// TIA Portal V20 export
FUNCTION_BLOCK "LER_InspectionInterface"   // FB50060, LAD
// stored: Access Published, MemoryReserve 100, SetENOAutomatically false
   VAR_INPUT
      Clamped : Bool;
      UnClamped : Bool;
      Celldetect : Bool;
      DryRun : Bool;
      SoftCam_X : "LER_typeSoftCamInterface";   // [6] Avoid , [7] Inst contac,[1]Ready
      SoftCam_Z : "LER_typeSoftCamInterface";   // [1] Ready , Avoid
      SoftCAm_C : "LER_typeSoftCamInterface";
      ProductionTimeTriger : Bool;
      Part_ID : String[32];
   END_VAR
   VAR_OUTPUT
      Axis_DisChargePositionLock : Bool;
      Axis_DisChargePositionCmd : Bool;   // for AutoSeq
      Axis_AvoidPositionCmd : Bool;   // for AutoSeq
      Axis_LoadComeplte : Bool;
      Insp_Req_Unclamp : Bool;   // for AutoSeq
   END_VAR
   VAR_IN_OUT
      BA60 : "LER_typeCommunicationInspection";
   END_VAR
   VAR
      DTL : DTL;
      STKtoINSP_Log : Array[0..50] of "LER_typeCommonDataInspection";
      P : Array[0..15] of Bool;
      Logic : Struct
         "a" : Bool;
         "b" : Bool;
      END_STRUCT;
      CleanData : "LER_typeCommonDataInspection";
   END_VAR
   VAR_TEMP
      REt : Int;
   END_VAR
   VAR_TEMP   // added for the SCL form of the ladder/FBD networks
      _w1 : Bool;
   END_VAR
BEGIN

REGION Network 2
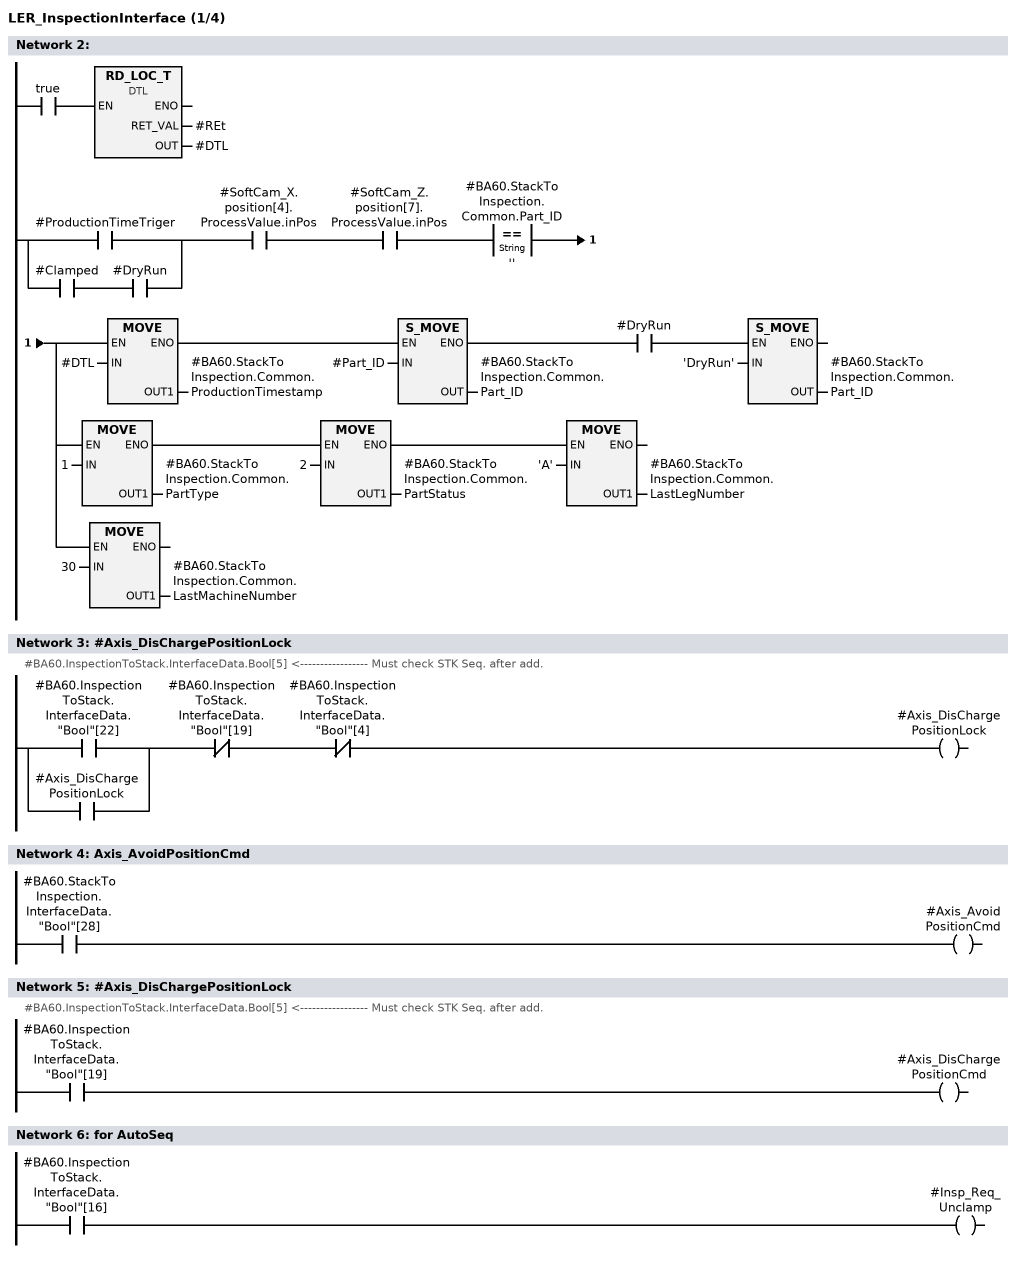
   RUNG wire#powerrail
      Contact( true )
      { S7_Templates := "date_type := DTL" } RD_LOC_T(RET_VAL => #REt, OUT => #DTL)
   END_RUNG
   RUNG wire#powerrail
      Contact( #ProductionTimeTriger )
      wire#w1
      Contact( #SoftCam_X.position[4].ProcessValue.inPos )
      Contact( #SoftCam_Z.position[7].ProcessValue.inPos )
      { S7_Templates := "SrcType := String" } EQ_Contact(in1 := #BA60.StackToInspection.Common.Part_ID, in2 := '')
      wire#w2
      Move(in := #DTL, out1 => #BA60.StackToInspection.Common.ProductionTimestamp)
      S_Move(in := #Part_ID, out => #BA60.StackToInspection.Common.Part_ID)
      Contact( #DryRun )
      S_Move(in := 'DryRun', out => #BA60.StackToInspection.Common.Part_ID)
   END_RUNG
   RUNG wire#powerrail
      Contact( #Clamped )
      Contact( #DryRun )
   END_RUNG wire#w1
   RUNG wire#w2
      Move(in := 1, out1 => #BA60.StackToInspection.Common.PartType)
      Move(in := 2, out1 => #BA60.StackToInspection.Common.PartStatus)
      Move(in := 'A', out1 => #BA60.StackToInspection.Common.LastLegNumber)
   END_RUNG
   RUNG wire#w2
      Move(in := 30, out1 => #BA60.StackToInspection.Common.LastMachineNumber)
   END_RUNG
   // the same network as SCL:
   IF true THEN #REt := RD_LOC_T(OUT => #DTL); END_IF;
   #_w1 := (#ProductionTimeTriger OR (#Clamped AND #DryRun)) AND #SoftCam_X.position[4].ProcessValue.inPos AND #SoftCam_Z.position[7].ProcessValue.inPos AND (#BA60.StackToInspection.Common.Part_ID = '');
   IF #_w1 THEN
       #BA60.StackToInspection.Common.ProductionTimestamp := #DTL;
       #BA60.StackToInspection.Common.Part_ID := #Part_ID;
   END_IF;
   IF #_w1 AND #DryRun THEN #BA60.StackToInspection.Common.Part_ID := 'DryRun'; END_IF;
   IF #_w1 THEN
       #BA60.StackToInspection.Common.PartType := 1;
       #BA60.StackToInspection.Common.PartStatus := 2;
       #BA60.StackToInspection.Common.LastLegNumber := 'A';
       #BA60.StackToInspection.Common.LastMachineNumber := 30;
   END_IF;
END_REGION

REGION Network 3: #Axis_DisChargePositionLock
   // #BA60.InspectionToStack.InterfaceData.Bool[5] <----------------- Must check STK Seq. after add.
   RUNG wire#powerrail
      Contact( #BA60.InspectionToStack.InterfaceData."Bool"[22] )
      wire#w1
      I_Contact( #BA60.InspectionToStack.InterfaceData."Bool"[19] )
      I_Contact( #BA60.InspectionToStack.InterfaceData."Bool"[4] )
      Coil( #Axis_DisChargePositionLock )
   END_RUNG
   RUNG wire#powerrail
      Contact( #Axis_DisChargePositionLock )
   END_RUNG wire#w1
   // the same network as SCL:
   #Axis_DisChargePositionLock := (#BA60.InspectionToStack.InterfaceData."Bool"[22] OR #Axis_DisChargePositionLock) AND NOT #BA60.InspectionToStack.InterfaceData."Bool"[19] AND NOT #BA60.InspectionToStack.InterfaceData."Bool"[4];
END_REGION

REGION Network 4: Axis_AvoidPositionCmd
   RUNG wire#powerrail
      Contact( #BA60.StackToInspection.InterfaceData."Bool"[28] )
      Coil( #Axis_AvoidPositionCmd )
   END_RUNG
   // the same network as SCL:
   #Axis_AvoidPositionCmd := #BA60.StackToInspection.InterfaceData."Bool"[28];
END_REGION

REGION Network 5: #Axis_DisChargePositionLock
   // #BA60.InspectionToStack.InterfaceData.Bool[5] <----------------- Must check STK Seq. after add.
   RUNG wire#powerrail
      Contact( #BA60.InspectionToStack.InterfaceData."Bool"[19] )
      Coil( #Axis_DisChargePositionCmd )
   END_RUNG
   // the same network as SCL:
   #Axis_DisChargePositionCmd := #BA60.InspectionToStack.InterfaceData."Bool"[19];
END_REGION

REGION Network 6: for AutoSeq
   RUNG wire#powerrail
      Contact( #BA60.InspectionToStack.InterfaceData."Bool"[16] )
      Coil( #Insp_Req_Unclamp )
   END_RUNG
   // the same network as SCL:
   #Insp_Req_Unclamp := #BA60.InspectionToStack.InterfaceData."Bool"[16];
END_REGION

REGION Network 7: for AutoSeq - Load Complete
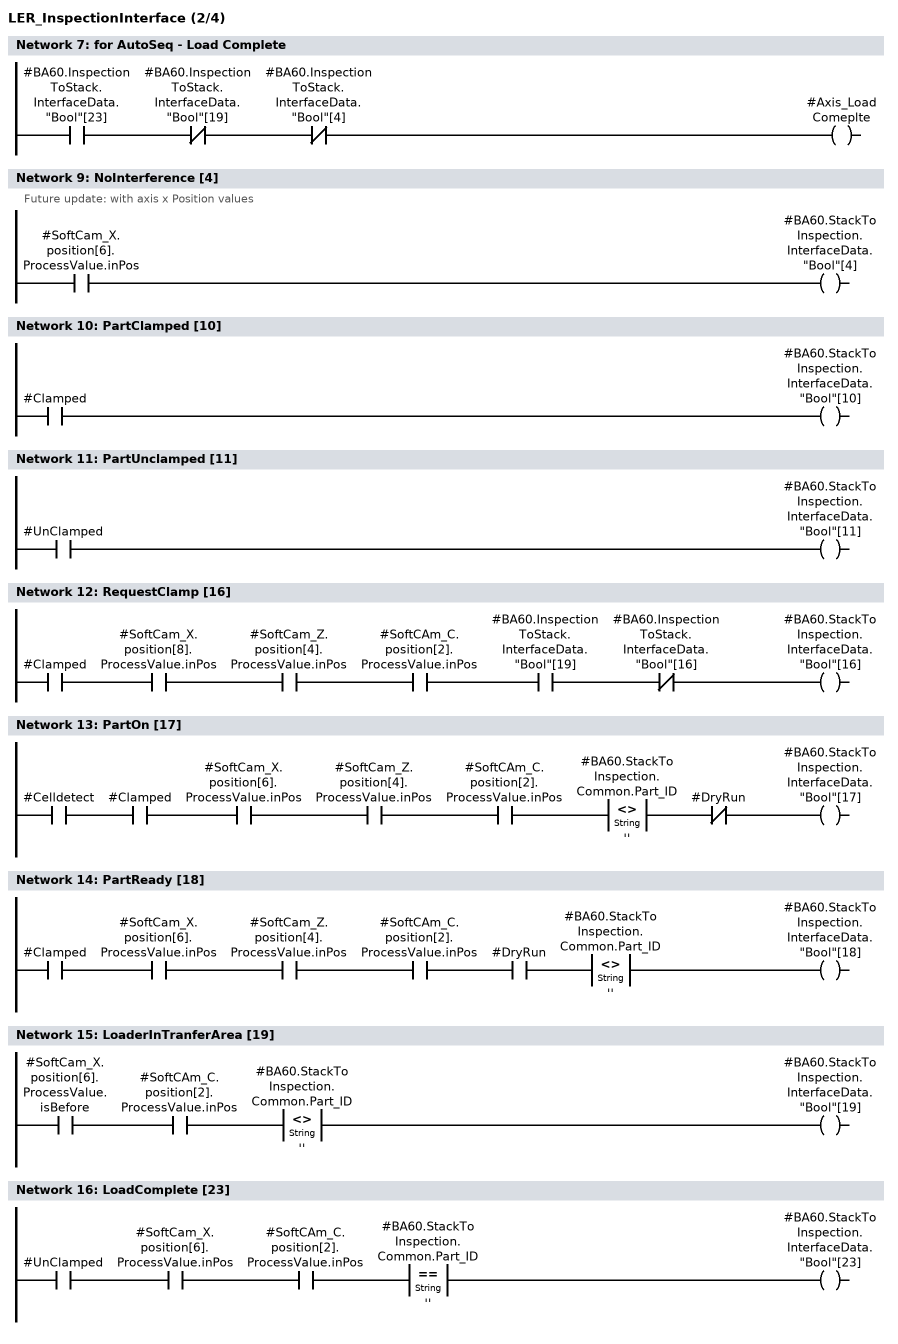
   RUNG wire#powerrail
      Contact( #BA60.InspectionToStack.InterfaceData."Bool"[23] )
      I_Contact( #BA60.InspectionToStack.InterfaceData."Bool"[19] )
      I_Contact( #BA60.InspectionToStack.InterfaceData."Bool"[4] )
      Coil( #Axis_LoadComeplte )
   END_RUNG
   // the same network as SCL:
   #Axis_LoadComeplte := #BA60.InspectionToStack.InterfaceData."Bool"[23] AND NOT #BA60.InspectionToStack.InterfaceData."Bool"[19] AND NOT #BA60.InspectionToStack.InterfaceData."Bool"[4];
END_REGION

REGION Network 8: ========================= Inspection To Stack ===================================
END_REGION

REGION Network 9: NoInterference [4]
   // Future update: with axis x Position values
   RUNG wire#powerrail
      Contact( #SoftCam_X.position[6].ProcessValue.inPos )
      Coil( #BA60.StackToInspection.InterfaceData."Bool"[4] )
   END_RUNG
   // the same network as SCL:
   #BA60.StackToInspection.InterfaceData."Bool"[4] := #SoftCam_X.position[6].ProcessValue.inPos;
END_REGION

REGION Network 10: PartClamped [10]
   RUNG wire#powerrail
      Contact( #Clamped )
      Coil( #BA60.StackToInspection.InterfaceData."Bool"[10] )
   END_RUNG
   // the same network as SCL:
   #BA60.StackToInspection.InterfaceData."Bool"[10] := #Clamped;
END_REGION

REGION Network 11: PartUnclamped [11]
   RUNG wire#powerrail
      Contact( #UnClamped )
      Coil( #BA60.StackToInspection.InterfaceData."Bool"[11] )
   END_RUNG
   // the same network as SCL:
   #BA60.StackToInspection.InterfaceData."Bool"[11] := #UnClamped;
END_REGION

REGION Network 12: RequestClamp [16]
   RUNG wire#powerrail
      Contact( #Clamped )
      Contact( #SoftCam_X.position[8].ProcessValue.inPos )
      Contact( #SoftCam_Z.position[4].ProcessValue.inPos )
      Contact( #SoftCAm_C.position[2].ProcessValue.inPos )
      Contact( #BA60.InspectionToStack.InterfaceData."Bool"[19] )
      I_Contact( #BA60.InspectionToStack.InterfaceData."Bool"[16] )
      Coil( #BA60.StackToInspection.InterfaceData."Bool"[16] )
   END_RUNG
   // the same network as SCL:
   #BA60.StackToInspection.InterfaceData."Bool"[16] := #Clamped AND #SoftCam_X.position[8].ProcessValue.inPos AND #SoftCam_Z.position[4].ProcessValue.inPos AND #SoftCAm_C.position[2].ProcessValue.inPos AND #BA60.InspectionToStack.InterfaceData."Bool"[19] AND NOT #BA60.InspectionToStack.InterfaceData."Bool"[16];
END_REGION

REGION Network 13: PartOn [17]
   RUNG wire#powerrail
      Contact( #Celldetect )
      Contact( #Clamped )
      Contact( #SoftCam_X.position[6].ProcessValue.inPos )
      Contact( #SoftCam_Z.position[4].ProcessValue.inPos )
      Contact( #SoftCAm_C.position[2].ProcessValue.inPos )
      { S7_Templates := "SrcType := String" } NE_Contact(in1 := #BA60.StackToInspection.Common.Part_ID, in2 := '')
      I_Contact( #DryRun )
      Coil( #BA60.StackToInspection.InterfaceData."Bool"[17] )
   END_RUNG
   // the same network as SCL:
   #BA60.StackToInspection.InterfaceData."Bool"[17] := #Celldetect AND #Clamped AND #SoftCam_X.position[6].ProcessValue.inPos AND #SoftCam_Z.position[4].ProcessValue.inPos AND #SoftCAm_C.position[2].ProcessValue.inPos AND (#BA60.StackToInspection.Common.Part_ID <> '') AND NOT #DryRun;
END_REGION

REGION Network 14: PartReady [18]
   RUNG wire#powerrail
      Contact( #Clamped )
      Contact( #SoftCam_X.position[6].ProcessValue.inPos )
      Contact( #SoftCam_Z.position[4].ProcessValue.inPos )
      Contact( #SoftCAm_C.position[2].ProcessValue.inPos )
      Contact( #DryRun )
      { S7_Templates := "SrcType := String" } NE_Contact(in1 := #BA60.StackToInspection.Common.Part_ID, in2 := '')
      Coil( #BA60.StackToInspection.InterfaceData."Bool"[18] )
   END_RUNG
   // the same network as SCL:
   #BA60.StackToInspection.InterfaceData."Bool"[18] := #Clamped AND #SoftCam_X.position[6].ProcessValue.inPos AND #SoftCam_Z.position[4].ProcessValue.inPos AND #SoftCAm_C.position[2].ProcessValue.inPos AND #DryRun AND (#BA60.StackToInspection.Common.Part_ID <> '');
END_REGION

REGION Network 15: LoaderInTranferArea [19]
   RUNG wire#powerrail
      Contact( #SoftCam_X.position[6].ProcessValue.isBefore )
      Contact( #SoftCAm_C.position[2].ProcessValue.inPos )
      { S7_Templates := "SrcType := String" } NE_Contact(in1 := #BA60.StackToInspection.Common.Part_ID, in2 := '')
      Coil( #BA60.StackToInspection.InterfaceData."Bool"[19] )
   END_RUNG
   // the same network as SCL:
   #BA60.StackToInspection.InterfaceData."Bool"[19] := #SoftCam_X.position[6].ProcessValue.isBefore AND #SoftCAm_C.position[2].ProcessValue.inPos AND (#BA60.StackToInspection.Common.Part_ID <> '');
END_REGION

REGION Network 16: LoadComplete [23]
   RUNG wire#powerrail
      Contact( #UnClamped )
      Contact( #SoftCam_X.position[6].ProcessValue.inPos )
      Contact( #SoftCAm_C.position[2].ProcessValue.inPos )
      { S7_Templates := "SrcType := String" } EQ_Contact(in1 := #BA60.StackToInspection.Common.Part_ID, in2 := '')
      Coil( #BA60.StackToInspection.InterfaceData."Bool"[23] )
   END_RUNG
   // the same network as SCL:
   #BA60.StackToInspection.InterfaceData."Bool"[23] := #UnClamped AND #SoftCam_X.position[6].ProcessValue.inPos AND #SoftCAm_C.position[2].ProcessValue.inPos AND (#BA60.StackToInspection.Common.Part_ID = '');
END_REGION

REGION Network 17: DataCatchUp [26]
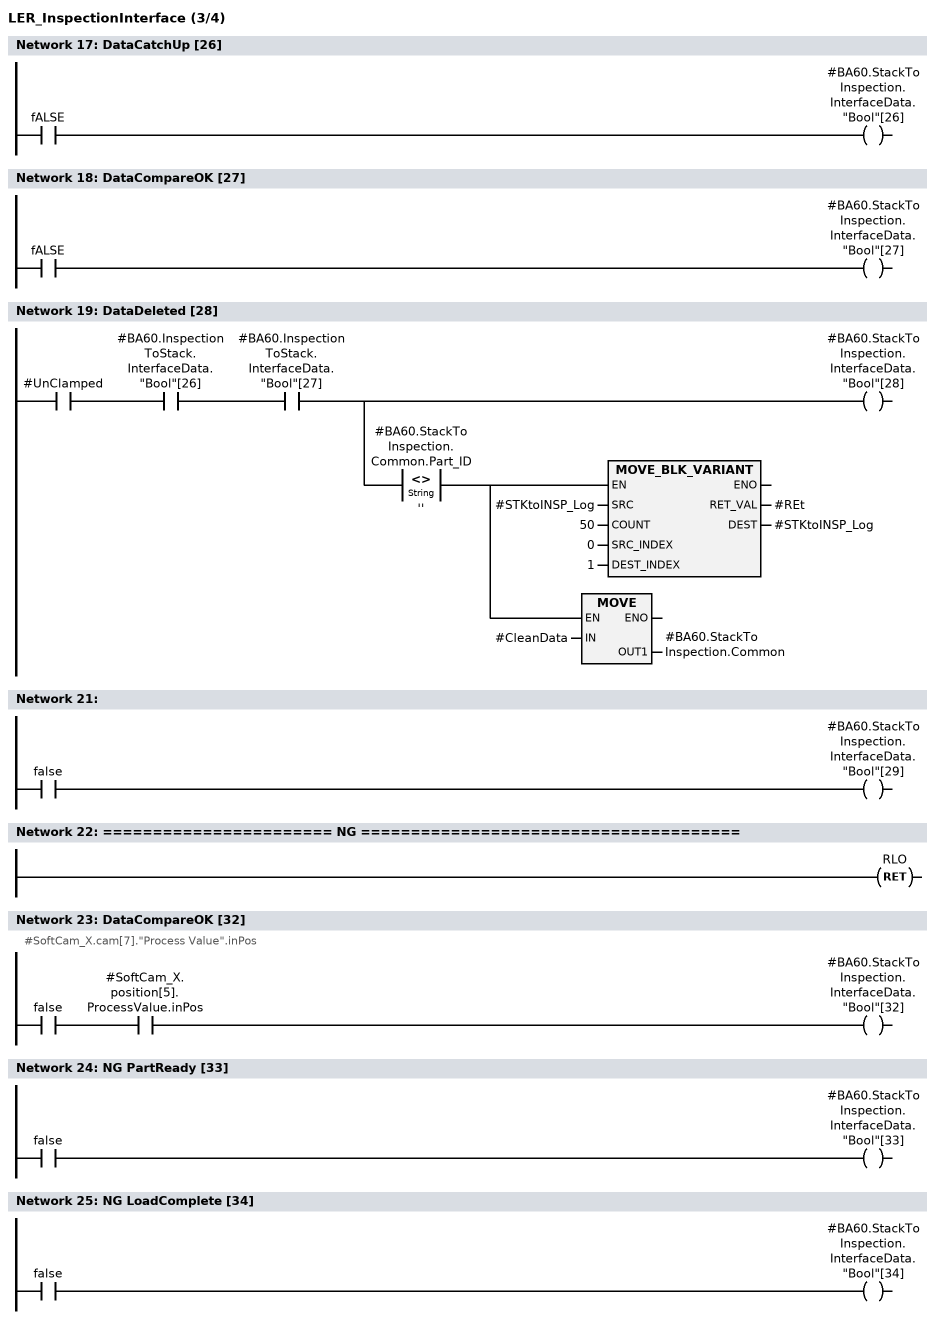
   RUNG wire#powerrail
      Contact( fALSE )
      Coil( #BA60.StackToInspection.InterfaceData."Bool"[26] )
   END_RUNG
   // the same network as SCL:
   #BA60.StackToInspection.InterfaceData."Bool"[26] := fALSE;
END_REGION

REGION Network 18: DataCompareOK [27]
   RUNG wire#powerrail
      Contact( fALSE )
      Coil( #BA60.StackToInspection.InterfaceData."Bool"[27] )
   END_RUNG
   // the same network as SCL:
   #BA60.StackToInspection.InterfaceData."Bool"[27] := fALSE;
END_REGION

REGION Network 19: DataDeleted [28]
   RUNG wire#powerrail
      Contact( #UnClamped )
      Contact( #BA60.InspectionToStack.InterfaceData."Bool"[26] )
      Contact( #BA60.InspectionToStack.InterfaceData."Bool"[27] )
      wire#w1
      Coil( #BA60.StackToInspection.InterfaceData."Bool"[28] )
   END_RUNG
   RUNG wire#w1
      { S7_Templates := "SrcType := String" } NE_Contact(in1 := #BA60.StackToInspection.Common.Part_ID, in2 := '')
      wire#w2
      MOVE_BLK_VARIANT(SRC := #STKtoINSP_Log, COUNT := 50, SRC_INDEX := 0, DEST_INDEX := 1, Ret_Val => #REt, DEST => #STKtoINSP_Log)
   END_RUNG
   RUNG wire#w2
      Move(in := #CleanData, out1 => #BA60.StackToInspection.Common)
   END_RUNG
   // the same network as SCL:
   #BA60.StackToInspection.InterfaceData."Bool"[28] := #UnClamped AND #BA60.InspectionToStack.InterfaceData."Bool"[26] AND #BA60.InspectionToStack.InterfaceData."Bool"[27];
   IF #UnClamped AND #BA60.InspectionToStack.InterfaceData."Bool"[26] AND #BA60.InspectionToStack.InterfaceData."Bool"[27] AND (#BA60.StackToInspection.Common.Part_ID <> '') THEN
       #REt := MOVE_BLK_VARIANT(SRC := #STKtoINSP_Log,
                               COUNT := 50,
                               SRC_INDEX := 0,
                               DEST_INDEX := 1,
                               DEST => #STKtoINSP_Log);
       #BA60.StackToInspection.Common := #CleanData;
   END_IF;
END_REGION

REGION Network 21
   RUNG wire#powerrail
      Contact( false )
      Coil( #BA60.StackToInspection.InterfaceData."Bool"[29] )
   END_RUNG
   // the same network as SCL:
   #BA60.StackToInspection.InterfaceData."Bool"[29] := false;
END_REGION

REGION Network 22: ======================= NG ======================================
   ENO := TRUE;
   RETURN;
END_REGION

REGION Network 23: DataCompareOK [32]
   // #SoftCam_X.cam[7]."Process Value".inPos
   RUNG wire#powerrail
      Contact( false )
      Contact( #SoftCam_X.position[5].ProcessValue.inPos )
      Coil( #BA60.StackToInspection.InterfaceData."Bool"[32] )
   END_RUNG
   // the same network as SCL:
   #BA60.StackToInspection.InterfaceData."Bool"[32] := false AND #SoftCam_X.position[5].ProcessValue.inPos;
END_REGION

REGION Network 24: NG PartReady [33]
   RUNG wire#powerrail
      Contact( false )
      Coil( #BA60.StackToInspection.InterfaceData."Bool"[33] )
   END_RUNG
   // the same network as SCL:
   #BA60.StackToInspection.InterfaceData."Bool"[33] := false;
END_REGION

REGION Network 25: NG LoadComplete [34]
   RUNG wire#powerrail
      Contact( false )
      Coil( #BA60.StackToInspection.InterfaceData."Bool"[34] )
   END_RUNG
   // the same network as SCL:
   #BA60.StackToInspection.InterfaceData."Bool"[34] := false;
END_REGION

REGION Network 26: ReturnToHome [46]
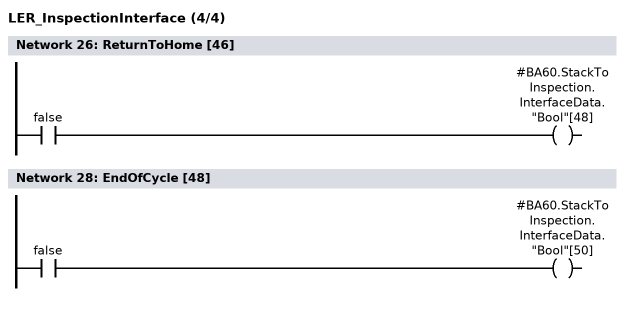
   RUNG wire#powerrail
      Contact( false )
      Coil( #BA60.StackToInspection.InterfaceData."Bool"[48] )
   END_RUNG
   // the same network as SCL:
   #BA60.StackToInspection.InterfaceData."Bool"[48] := false;
END_REGION

REGION Network 27: AutoStart [47]
END_REGION

REGION Network 28: EndOfCycle [48]
   RUNG wire#powerrail
      Contact( false )
      Coil( #BA60.StackToInspection.InterfaceData."Bool"[50] )
   END_RUNG
   // the same network as SCL:
   #BA60.StackToInspection.InterfaceData."Bool"[50] := false;
END_REGION

REGION Network 29: NG RequestClamp [49]
END_REGION

REGION Network 30: ======================= State MAnager Status ======================================
END_REGION
END_FUNCTION_BLOCK
